{attribute 'linkalways'} 
{attribute 'no_explicit_call' := 'This FB is a CLASS and must be accessed using methods or properties'}
{attribute 'enable_dynamic_creation'}
FUNCTION_BLOCK Node_F_VN_GetImageWidth EXTENDS VisionNode
VAR
    ipImage : _ITcVnImage;
    nWidth : _UDINT(0);
    hrPrev : _HRESULT(S_OK);
	hresult : _HRESULT(S_OK);
END_VAR

METHOD PUBLIC  Clone : I_Node
VAR
	pNode : POINTER TO Node_F_VN_GetImageWidth;
END_VAR
pNode := __NEW(Node_F_VN_GetImageWidth);
Clone := pNode^;
END_METHOD

METHOD FB_init : BOOL
VAR_INPUT
	bInitRetains : BOOL; // if TRUE, the retain variables are initialized (warm start / cold start)
	bInCopyCode : BOOL;  // if TRUE, the instance afterwards gets moved into the copy code (online change)
END_VAR
AddInput('ipImage', ipImage);
AddInput('hrPrev', hrPrev);
AddOutput('nWidth', nWidth);
AddOutput('hresult',hresult);
END_METHOD

METHOD PROTECTED OnExecute : HRESULT
hresult.Value := F_VN_GetImageWidth(
    ipImage := ipImage.Value,
    nWidth := nWidth.Value,
	hrPrev:= hrPrev.Value);
END_METHOD

METHOD PUBLIC PreExecutionCheck
VAR_INPUT
	Check : I_PreExecutionChecks;
END_VAR
IF FAILED(hrPrev.Value) THEN
    RETURN;
END_IF

Check.IsTrue(ipImage.IsValid, 'ipImage must contain an image');
END_METHOD

END_FUNCTION_BLOCK

(* stored: Version 1.1.0.1, ProductVersion 3.1.4024.13
   POU Node_F_VN_GetImageWidth: Id {e9758da4-c4e5-0ffb-2402-ff08a2bc031b}, SpecialFunc None
   Folder Constructor: Id {1fb21175-74f5-04f6-0ac9-9abd9a2d47c6}
   Method Clone: Id {1672303e-602a-0128-0396-e42241f9ab7d}
   Method FB_init: Id {38d4903c-d9e2-000a-303e-ba346f3a9e39}
   Method OnExecute: Id {ee3bb618-d9a4-0da1-0a26-f3c6850f1bef}
   Method PreExecutionCheck: Id {192ad020-23d2-09e0-1fce-1b0f76ccb428} *)
